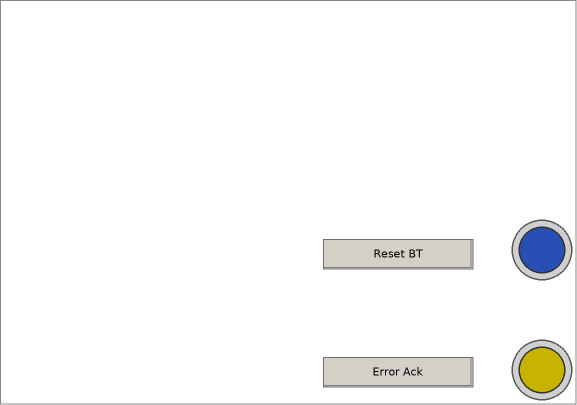
VISUALIZATION Visualization  // 577x405
    Button (323,239 150x30), "Reset BT", pressed state: GVL_Safety.bResetButtonVISU
        OnMouseClick: toggle GVL_Safety.bResetButtonVISU
    Lamp1 (507,215 70x70), variable: GVL_Safety.bResetButtonVISU, style: Lamp-Lamp1-Blue
    Button (323,357 150x30), "Error Ack", pressed state: GVL_Safety.bAckButtonVISU
        OnMouseClick: toggle GVL_Safety.bAckButtonVISU
    Lamp1 (507,335 70x70), variable: GVL_Safety.bSafetyErrorAck, style: Lamp-Lamp1-Yellow
END_VISUALIZATION

(* stored: Version 1.1.0.1, ProductVersion 3.1.4024.12
   Visu Visualization: Id {9245dd2e-88c7-4ebc-942a-b09707f3c1ca} *)
